FUNCTION_BLOCK PUBLIC FB_ModeControlBox IMPLEMENTS I_Mode
VAR_INPUT
END_VAR
VAR_OUTPUT
END_VAR
VAR
END_VAR

METHOD Auto
VAR_INPUT
	bEnable	: BOOL;
END_VAR
IF bEnable THEN
Outputs.fCylinderPosition := CraneSimulation.fPositionAutoMode;
Outputs.eMode := E_Mode.Auto; 
END_IF
END_METHOD

METHOD Manual
VAR_INPUT
	bEnable	: BOOL;
END_VAR
IF bEnable THEN
Outputs.fCylinderPosition := HMI.fManualCylinderPositionReference;
Outputs.eMode := E_Mode.Manual;
END_IF
END_METHOD

METHOD Off
VAR_INPUT
	bEnable	: BOOL;
END_VAR
IF bEnable THEN
Outputs.fCylinderPosition := 0;
Outputs.eMode := E_Mode.Off; 
END_IF
END_METHOD

END_FUNCTION_BLOCK

(* stored: Version 1.1.0.1, ProductVersion 3.1.4024.10
   POU FB_ModeControlBox: Id {7ddd8f23-6d80-4096-b07f-1e70525896a4}, SpecialFunc None
   Method Auto: Id {48682564-9766-49f3-bf8b-f40af20c1211}
   Method Manual: Id {1d156ece-8246-40d7-b076-905685867dca}
   Method Off: Id {6d2093be-f10c-4755-a701-cd935c7e21b0} *)
